// TIA Portal project "Conveyor_System" (V15.1)

(* hardware
DEVICE "S7-1200 station_1"  S7-1200 Station
   slot 0: "Rack_0"  S7-1200 Rack  Rack  V1.0
   slot 1: "PLC_1"  CPU 1214C DC/DC/DC  6ES7 214-1AG40-0XB0  V4.2
DEVICE "HMI_1"  KTP700 Basic PN
   slot 0: "HMI_1"  KTP700 Basic PN  6AV2 123-2GB03-0AX0  15.1.0.0
   slot 1: "HMI_RT_1"  KTP700 Basic PN  6AV2 123-2GB03-0AX0  15.1.0.0
   slot 5: "HMI_1.IE_CP_1"  PROFINET Interface  15.0.1.0
      slot 1: "PROFINET Interface_1"  PROFINET Interface
         slot 1: "Port_1"  Port
*)

// ===== PLC "PLC_1"  CPU 1214C DC/DC/DC =====

VAR_GLOBAL   // PLC tag table "Default tag table"
   "START" AT %M0.0 : Bool;
   "STOP" AT %M0.1 : Bool;
   "RESET" AT %M0.2 : Bool;
   "BFULL" AT %M0.3 : Bool;
   "BCHANGE" AT %M0.4 : Bool;
   "BSENSOR" AT %M0.5 : Bool;
   "SYSTEM_I" AT %M0.6 : Bool;
   "SYSTEM_II" AT %M0.7 : Bool;
   "SYSTEM_III" AT %M1.0 : Bool;
   "SENSOR_I" AT %M1.1 : Bool;
   "SENSOR_II" AT %M1.2 : Bool;
   "CT_DONE_I" AT %M1.3 : Bool;
   "CT_DONE_II" AT %M1.4 : Bool;
   "CT_I" AT %M1.5 : Bool;
   "CT_II" AT %M1.6 : Bool;
   "mTimerSystem3" AT %M1.7 : Bool;
END_VAR

// folder: System blocks/Program resources

DATA_BLOCK "IEC_Counter_0_DB_1"   // DB1
{ S7_Optimized_Access := 'TRUE' }
AUTHOR : Simatic
FAMILY : IEC
NAME : CNTR
VERSION : 1.0
// stored: InstanceOfName IEC_COUNTER
"IEC_COUNTER"
BEGIN
END_DATA_BLOCK

DATA_BLOCK "IEC_Counter_0_DB_2"   // DB2
{ S7_Optimized_Access := 'TRUE' }
AUTHOR : Simatic
FAMILY : IEC
NAME : CNTR
VERSION : 1.0
// stored: InstanceOfName IEC_COUNTER
"IEC_COUNTER"
BEGIN
END_DATA_BLOCK

DATA_BLOCK "IEC_Timer_0_DB"   // DB3
{ S7_Optimized_Access := 'TRUE' }
AUTHOR : Simatic
FAMILY : IEC
NAME : IEC_TMR
VERSION : 1.0
// stored: InstanceOfName IEC_TIMER
"IEC_TIMER"
BEGIN
END_DATA_BLOCK

DATA_BLOCK "IEC_Timer_0_DB_1"   // DB4
{ S7_Optimized_Access := 'TRUE' }
AUTHOR : Simatic
FAMILY : IEC
NAME : IEC_TMR
VERSION : 1.0
// stored: InstanceOfName IEC_TIMER
"IEC_TIMER"
BEGIN
END_DATA_BLOCK

// folder: (top level)

FUNCTION "ConveyorSystem_Function" : Void   // FC1, SCL
{ S7_Optimized_Access := 'TRUE' }
VERSION : 0.1
BEGIN
    REGION ALGORITMA



         // [ALGORITMA]

         // 1-START'a basıldığında sistem aktif olacak.
         // 2-Sistem1 ve Sistem2 çalışmaya başlayacak.
         // 3-Sistem1 üç tane, Sistem2 ise beş tane top sayacak.
         // 4-BOX dolduğunda, (3+5=8) BOX-FULL sensörü uyarı verecek.
         // 5-BOX-FULL uyarısı 3 saniye boyunca devam edecek.
         // 6-Uyarı sonunda BOX-FULL sensörü devre dışı kalacak.
         // 7-BOX-CHANGING sensörü devreye girecek ve Sistem3 çalışmaya başlayacak.
         // 8-Sistem3 beş saniye boyunca çalışacak.
         // 9-Sistem kendini başa alacak.

         // [NOTLAR]

         // 1-Kutu yerinde değilse, düşürüldüyse otomatik olarak sensör algısı ile stoplanacak.
         // 2-Kutu yerindeyse sistem kaldığı yerden çalışmaya devam edecek.
         // 3-Acil durum için Stop'a basıldığında sistem resetlenmeden kaldığı yerde durdurulacak.




   END_REGION


   IF "BSENSOR" THEN

       "SYSTEM_I" := TRUE;
       "SYSTEM_II" := TRUE;
       "BFULL" := FALSE;

   END_IF;


   IF NOT "BSENSOR" AND "START" THEN
       "SYSTEM_I" := FALSE;
       "SYSTEM_II" := FALSE;
       "BFULL" := FALSE;
       "CT_I" := FALSE;
       "CT_II" := FALSE;
   END_IF;


   IF NOT "BSENSOR"  THEN
       "SYSTEM_I" := FALSE;
       "SYSTEM_II" := FALSE;
       "START" := FALSE;
       "BFULL" := FALSE;
       "CT_I" := FALSE;
       "CT_II" := FALSE;
   END_IF;

   IF "BSENSOR" AND NOT "START" THEN
       "SYSTEM_I" := FALSE;
       "SYSTEM_II" := FALSE;
       "CT_I" := FALSE;
       "CT_II" := FALSE;
   END_IF;

   IF "BSENSOR" AND "START" THEN
       "SYSTEM_I" := TRUE;
       "SYSTEM_II" := TRUE;

   END_IF;


   "IEC_Counter_0_DB_1".CTU(CU := "CT_I" AND "IEC_Counter_0_DB_1".CV < 3 AND NOT "STOP",
                            R := "RESET",
                            PV := 3,
                            Q => "CT_DONE_I");

   "IEC_Counter_0_DB_2".CTU(CU := "CT_II" AND "IEC_Counter_0_DB_2".CV < 5 AND NOT "STOP",
                            R := "RESET",
                            PV := 5,
                            Q => "CT_DONE_II");


   IF "RESET" THEN
       "BFULL" := FALSE;
   END_IF;


   IF "STOP" THEN
       "SYSTEM_I" := FALSE;
       "SYSTEM_II" := FALSE;
       "SYSTEM_III" := FALSE;


   END_IF;
   IF "CT_DONE_I" AND "CT_DONE_II" THEN

       "BFULL" := TRUE;

   END_IF;



   "IEC_Timer_0_DB".TON(IN := "BFULL",
                       PT := T#5S);
   IF "IEC_Timer_0_DB".Q THEN
       "SYSTEM_III" := TRUE;
       "BCHANGE" := TRUE;
       "RESET" := TRUE;
       "mTimerSystem3" := true;
   END_IF;


       "IEC_Timer_0_DB_1".TON(IN := "mTimerSystem3",
                             PT := T#5S);
       IF "IEC_Timer_0_DB_1".Q THEN
           "mTimerSystem3" := FALSE;
           "SYSTEM_III" := FALSE;
           "RESET" := FALSE;
           "BCHANGE" := FALSE;
           "BFULL" := FALSE;
       END_IF;
END_FUNCTION

ORGANIZATION_BLOCK "Main"   // OB1, LAD, ProgramCycle
TITLE = "Main Program Sweep (Cycle)"
{ S7_Optimized_Access := 'TRUE' }
VERSION : 0.1
   VAR_INPUT
      Initial_Call : Bool;   // Initial call of this OB
      Remanence : Bool;   // =True, if remanent data are available
   END_VAR
BEGIN

REGION Network 1
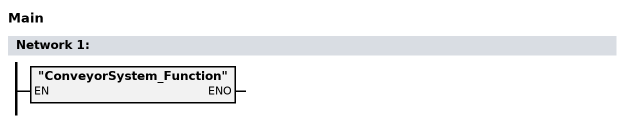
   RUNG wire#powerrail
      "ConveyorSystem_Function"()
   END_RUNG
   // the same network as SCL:
   "ConveyorSystem_Function"();
END_REGION
END_ORGANIZATION_BLOCK

(* ===== HMI "HMI_RT_1" =====
system functions are stored by id; their names below are inferred from use
connection "HMI_Connection_1": ETHERNET, SMART_S7_1200_OMS

HMI tags "Default tag table"
   "START" : Bool = PLC START AT %M0.0, 1 s
   "STOP" : Bool = PLC STOP AT %M0.1, 1 s
   "RESET" : Bool = PLC RESET AT %M0.2, 1 s
   "BSENSOR" : Bool = PLC BSENSOR AT %M0.5, 1 s
   "BFULL" : Bool = PLC BFULL AT %M0.3, 1 s
   "SYSTEM_I" : Bool = PLC SYSTEM_I AT %M0.6, 1 s
   "SYSTEM_II" : Bool = PLC SYSTEM_II AT %M0.7, 1 s
   "SYSTEM_III" : Bool = PLC SYSTEM_III AT %M1.0, 1 s
   "CT_DONE_I" : Bool = PLC CT_DONE_I AT %M1.3, 1 s
   "CT_DONE_II" : Bool = PLC CT_DONE_II AT %M1.4, 1 s
   "BCHANGE" : Bool = PLC BCHANGE AT %M0.4, 1 s
   "CT_I" : Bool = PLC CT_I AT %M1.5, 1 s
   "CT_II" : Bool = PLC CT_II AT %M1.6, 1 s
   "IEC_Counter_0_DB_2_CV" : Int = PLC IEC_Counter_0_DB_2.CV, 1 s
   "IEC_Counter_0_DB_1_CV" : Int = PLC IEC_Counter_0_DB_1.CV, 1 s

Template "Template_1" 800x480
   Button "Exit" at 714,429 size 71x50; TextOff 'Exit'; PictureOff "ExitRuntime_KTP700_Basic_PN_TR"; PictureOn "ExitRuntime_KTP700_Basic_PN_TR"
      on Release: StopRuntime(0)
   Button "Template_Button" at 614,429 size 71x50; TextOff 'Text'
   Button "Template_Button_1" at 514,429 size 71x50; TextOff 'Text'
   Button "Template_Button_2" at 414,429 size 71x50; TextOff 'Text'
   Button "Template_Button_3" at 314,429 size 71x50; TextOff 'Text'
   Button "Template_Button_4" at 214,429 size 71x50; TextOff 'Text'
   Button "Alarms" at 114,429 size 71x50; TextOff 'Alarms'; PictureOff "AlarmDisplay_KTP700_Basic_PN_TR"; PictureOn "AlarmDisplay_KTP700_Basic_PN_TR"
      on Release: function_ef3f5d25("Alarm window_Unacknowledged", -1)
   Button "Start screen" at 14,429 size 71x50; TextOff 'Start screen'; PictureOff "NavigateHome_KTP700_Basic_PN_TR"; PictureOn "NavigateHome_KTP700_Basic_PN_TR"
      on Release: ActivateScreen("HMI Panel", 0)
   SymbolicIOField "Symbolic_IO_Field_Screen" at 93,9 size 600x33; TextOff '0'; TextOn '1'; TextList "TextList_ScreenNames"
   DateTimeField "HmiScreenItemData" at 695,25 size 105x25
   DateTimeField "HmiScreenItemData_1" at 695,0 size 105x25
   GraphicView "Logo" at 0,0 size 91x51; Picture "Logo of HMI_1"

screen "HMI Panel" 800x480, template "Template_1"
   Rectangle "Rectangle_3" at 26,296 size 274x40
      Appearance <- "SYSTEM_III"
   Button "Button_1" at 575,100 size 55x21; TextOff 'START'
      Appearance <- "START"
      on Press: InvertBit("START"); ResetBit("STOP")
   Button "Button_2" at 644,100 size 55x21; TextOff 'STOP'
      on Press: InvertBit("STOP"); ResetBit("START")
      Appearance <- "STOP"
   Button "Button_3" at 710,101 size 55x21; TextOff 'RESET'
      on Press: function_b14e0dd5("RESET", 0)
   Rectangle "Rectangle_5" at 463,222 size 56x19
      Appearance <- "BFULL"
   TextField "Text field_1" at 463,224 size 55x15; Text 'BOX FULL'
   TextField "Text field_4" at 308,306 size 73x18; Text 'SYSTEM-III'
   Rectangle "Rectangle_6" at 440,371 size 100x23
      Appearance <- "BCHANGE"
   TextField "Text field_5" at 440,375 size 100x15; Text 'BOX IS CHANGING'
   Button "Button_4" at 459,149 size 32x21; TextOff 'S-2'
      on Press: function_b14e0dd5("CT_II", 0)
   Button "Button_5" at 459,103 size 32x21; TextOff 'S-1'
      on Press: function_b14e0dd5("CT_I", 0)
   Button "Button_7" at 576,132 size 55x21; TextOff 'BOX SENSOR'
      on Press: InvertBit("BSENSOR")
      Appearance <- "BSENSOR"
   IOField "I/O field_3" at 386,98 size 57x32; FormatPattern 9; Unit  pcs
      ProcessValue <- "IEC_Counter_0_DB_1_CV"
   IOField "I/O field_1" at 386,145 size 57x32; FormatPattern 9; Unit  pcs
      ProcessValue <- "IEC_Counter_0_DB_2_CV"
   Bar "Bar_1" at 26,142 size 271x38; MinimumValue 0
      ProcessValue <- "IEC_Counter_0_DB_2_CV"
   Bar "Bar_2" at 26,94 size 271x38; MinimumValue 0; MaximumValue 3
      ProcessValue <- "IEC_Counter_0_DB_1_CV"
   TextField "Text field_2" at 300,104 size 63x18; Text 'SYSTEM-I'
   TextField "Text field_3" at 300,151 size 68x18; Text 'SYSTEM-II'
   TextField "Text field_6" at 286,7 size 254x34; Text 'CONVEYOR SYSTEM'
*)